{attribute addProperty BoxType "AX8206-0000-0102-0102"}
{attribute addProperty Id "Position_actual_value_invalidAT %I*BOOL812_1st_Additional_position_actual_value_invalidAT %I*BOOL813Ch_B_StatuswordAT %I*UINT1620Ch_B_Position_actual_valueAT %I*DINT3240"}
{attribute addProperty CRC "3044970419"}
{attribute addProperty SizeInBites "64"}
{attribute addProperty SizeInBytes "8"}
TYPE Ch_B_AxisMain_Inputs_B57E8FB3 :
STRUCT
	{attribute addProperty Name "Position_actual_value_invalid"}
	Position_actual_value_invalid AT %I* : BOOL;
	{attribute addProperty Name "_1st_Additional_position_actual_value_invalid"}
	_1st_Additional_position_actual_value_invalid AT %I* : BOOL;
	{attribute addProperty Name "Ch_B_Statusword"}
	Ch_B_Statusword AT %I* : UINT;
	{attribute addProperty Name "Ch_B_Position_actual_value"}
	Ch_B_Position_actual_value AT %I* : DINT;
END_STRUCT
END_TYPE

(* stored: Version 1.2.0.0, ProductVersion 3.1.4024.9
   DUT Ch_B_AxisMain_Inputs_B57E8FB3: Id {4c2105ba-71ad-4760-903c-143b644d6b86} *)
